(* PLC project PLC_DEV.project, CODESYS CODESYS V3.5 SP21 Patch 4 *)
(* stored: creationDateTime 1970-01-01T00:00:00, modificationDateTime 1970-01-01T00:00:00 *)

TYPE ST_IO_IN : STRUCT
  StartPB : BOOL;
  StopPB : BOOL;
  EStop : BOOL;
  LS_Extended : BOOL;
  LS_Retracted : BOOL;
  MotorFB : BOOL;
  TankLevel : REAL;  (* 0..100 % *)
  Pressure : REAL;
  ValvePosFB : REAL;  (* 0..100 % *)
END_STRUCT;
END_TYPE

TYPE ST_IO_OUT : STRUCT
  MotorRun : BOOL;
  Pump : BOOL;
  CylExtend : BOOL;
  CylRetract : BOOL;
  ValveCmd : REAL;  (* 0..100 % *)
  VFD_SpeedCmd : REAL;  (* 0..100 % *)
END_STRUCT;
END_TYPE

TYPE ST_IO : STRUCT
  In : ST_IO_IN;
  Out : ST_IO_OUT;
END_STRUCT;
END_TYPE

(* values of E_SIM_BOOL_MODE: FIXED: always FixedValue (or OverrideValue); TOGGLE: flips true/false every ChangeEvery; PULSE: true for PulseWidth every ChangeEvery *)

TYPE E_SIM_BOOL_MODE : (FIXED, TOGGLE, PULSE);
END_TYPE

(* values of E_SIM_INT_MODE: FIXED: fixed value; RAMP: add Increment every ChangeEvery; RANDOM: pseudo-random in range every ChangeEvery *)

TYPE E_SIM_INT_MODE : (FIXED, RAMP, RANDOM);
END_TYPE

TYPE E_RunMode : (DEV, STG, PROD);
END_TYPE

PROGRAM PLC_PRG
  VAR
    Boot : FB_ModeBoot;
    IOMan : FB_IO_Manager;
  END_VAR

                  // 1) Read ENV ONCE
Boot();

// 2) Route IO
IOMan(Mode := gMode, IO := gIO);

// 3) Control logic


// ---------------- Control Logic ----------------
IF gIO.In.EStop THEN
    gIO.Out.MotorRun := FALSE;
    gIO.Out.Pump := FALSE;
    gIO.Out.CylExtend := FALSE;
	gIO.Out.VFD_SpeedCmd := 0.0; // going back to 0
    gIO.Out.ValveCmd := 0.0;  // same here
ELSE
    IF gIO.In.StartPB THEN
        gIO.Out.MotorRun := TRUE;
        gIO.Out.Pump := TRUE;
        gIO.Out.VFD_SpeedCmd := 75.0; // Increase the speed 
        gIO.Out.ValveCmd := 15.0; // Valve command should be 15
    END_IF

    IF gIO.In.StopPB THEN
        gIO.Out.MotorRun := FALSE;
        gIO.Out.Pump := FALSE;
        gIO.Out.VFD_SpeedCmd := 0.0;
        gIO.Out.ValveCmd := 0.0;
    END_IF

    gIO.Out.CylExtend := gIO.Out.MotorRun;
    gIO.Out.CylRetract := NOT gIO.Out.MotorRun;
END_IF
                
END_PROGRAM

FUNCTION_BLOCK FB_IO_Prod
  VAR_IN_OUT
    IO : ST_IO;
  END_VAR

                  // ================= READ PROD INPUTS =================
// Map your physical / fieldbus / Modbus / MQTT inputs here
// Example:
// IO.In.StartPB      := TRUE;
// IO.In.StopPB       := DI_StopPB;
// IO.In.EStop        := DI_EStop;
// IO.In.LS_Extended  := DI_LS_Extended;
// IO.In.LS_Retracted := DI_LS_Retracted;
// IO.In.MotorFB      := DI_MotorFB;
//
// IO.In.TankLevel    := AI_TankLevel;
// IO.In.Pressure     := AI_Pressure;
// IO.In.ValvePosFB   := AI_ValvePosFB;

// ================= WRITE PROD OUTPUTS =================
// Example:
// DO_MotorRun     := IO.Out.MotorRun;
// DO_Pump         := IO.Out.Pump;
// DO_CylExtend    := IO.Out.CylExtend;
// DO_CylRetract   := IO.Out.CylRetract;
//
// AO_ValveCmd     := IO.Out.ValveCmd;
// AO_VFD_SpeedCmd := IO.Out.VFD_SpeedCmd;
                
END_FUNCTION_BLOCK

FUNCTION_BLOCK FB_IO_Manager
  VAR_INPUT
    Mode : E_RunMode;
  END_VAR
  VAR_IN_OUT
    IO : ST_IO;
  END_VAR
  VAR
    Sim : FB_IO_SIM;
    Prod : FB_IO_PROD;
  END_VAR

                  // DEV + STG = simulated IO
IF (Mode = E_RunMode.DEV) OR (Mode = E_RunMode.STG) THEN
    Sim(IO := IO);
ELSE
    Prod(IO := IO);
END_IF

                
END_FUNCTION_BLOCK

FUNCTION_BLOCK FB_ModeBoot
  VAR_OUTPUT
    Done : BOOL;
  END_VAR
  VAR
    init : BOOL;
    outBuf : STRING(64);
    res : DINT;
    n : DINT;
  END_VAR

                  IF Done THEN RETURN; END_IF
IF NOT init THEN
    init := TRUE;

    gMode := E_RunMode.PROD;   // safe default
    outBuf := '';

    n := SysProcessExecuteCommand2(
        pszCommand := '/usr/bin/head -c 4 /conf/codesyscontrol/env.txt',
        pszStdOut := outBuf,
        udiStdOutLen := SIZEOF(outBuf),
        pResult := ADR(res)
    );

    IF n >= 3 THEN
        IF (LEFT(outBuf, 3) = 'dev') OR (LEFT(outBuf, 3) = 'DEV') THEN
            gMode := E_RunMode.DEV;

        ELSIF (LEFT(outBuf, 3) = 'stg') OR (LEFT(outBuf, 3) = 'STG') THEN
            gMode := E_RunMode.STG;

        ELSIF (LEFT(outBuf, 4) = 'prod') OR (LEFT(outBuf, 4) = 'PROD') THEN
            gMode := E_RunMode.PROD;
        END_IF
    END_IF

    Done := TRUE;
END_IF


                
END_FUNCTION_BLOCK

FUNCTION_BLOCK FB_SimInt_Gen
  VAR_INPUT
    Enable : BOOL := TRUE;
    Mode : E_SIM_INT_MODE := E_SIM_INT_MODE.RAMP;
    MinValue : INT := 0;
    MaxValue : INT := 100;
    Increment : INT := 1;  (* used by RAMP *)
    ChangeEvery : TIME := TIME#200ms;
    Wrap : BOOL := TRUE;  (* RAMP behavior: wrap or clamp *)
    FixedValue : INT := 0;
    OverrideEn : BOOL := FALSE;
    OverrideValue : INT := 0;
  END_VAR
  VAR_OUTPUT
    Value : INT;
  END_VAR
  VAR
    tPeriod : TON;
    seedInt : INT := 12345;  (* random seed kept as INT only *)
    span : INT;
    nextVal : INT;
    tmp : INT;
  END_VAR

                  // ---------- guards ----------
IF NOT Enable THEN
    Value := MinValue;
    RETURN;
END_IF

IF OverrideEn THEN
    Value := OverrideValue;
    RETURN;
END_IF

IF MaxValue < MinValue THEN
    Value := MinValue;
    RETURN;
END_IF

// ---------- timing ----------
tPeriod(IN := TRUE, PT := ChangeEvery);
IF NOT tPeriod.Q THEN
    RETURN;
END_IF
tPeriod(IN := FALSE); // restart timer

// ---------- mode ----------
CASE Mode OF

E_SIM_INT_MODE.FIXED:
    Value := FixedValue;

E_SIM_INT_MODE.RAMP:
    nextVal := Value + Increment;

    IF Wrap THEN
        span := MaxValue - MinValue + 1;
        IF span <= 0 THEN span := 1; END_IF
        WHILE nextVal > MaxValue DO
            nextVal := nextVal - span;
        END_WHILE
        WHILE nextVal < MinValue DO
            nextVal := nextVal + span;
        END_WHILE
    ELSE
        IF nextVal > MaxValue THEN nextVal := MaxValue; END_IF
        IF nextVal < MinValue THEN nextVal := MinValue; END_IF
    END_IF

    Value := nextVal;

E_SIM_INT_MODE.RANDOM:
    // simple INT LCG (stays in INT domain)
    seedInt := seedInt * 109 + 89;

    // make it non-negative
    IF seedInt < 0 THEN
        seedInt := -seedInt;
    END_IF

    span := MaxValue - MinValue + 1;
    IF span <= 0 THEN span := 1; END_IF

    // reduce into 0..span-1 using subtraction (no MOD needed)
    tmp := seedInt;
    WHILE tmp >= span DO
        tmp := tmp - span;
    END_WHILE

    Value := MinValue + tmp;

END_CASE
                
END_FUNCTION_BLOCK

FUNCTION_BLOCK FB_SimBool_Gen
  VAR_INPUT
    Enable : BOOL := TRUE;
    Mode : E_SIM_BOOL_MODE := E_SIM_BOOL_MODE.TOGGLE;
    ChangeEvery : TIME := TIME#2s0ms;
    PulseWidth : TIME := TIME#150ms;
    FixedValue : BOOL := FALSE;
    OverrideEn : BOOL := FALSE;
    OverrideValue : BOOL := FALSE;
  END_VAR
  VAR_OUTPUT
    Value : BOOL;
  END_VAR
  VAR
    tPeriod : TON;
    tPulse : TON;
    state : BOOL := FALSE;
  END_VAR

                  IF NOT Enable THEN
    Value := FALSE;
    RETURN;
END_IF

IF OverrideEn THEN
    Value := OverrideValue;
    RETURN;
END_IF

CASE Mode OF

E_SIM_BOOL_MODE.FIXED:
    Value := FixedValue;

E_SIM_BOOL_MODE.TOGGLE:
    tPeriod(IN := TRUE, PT := ChangeEvery);
    IF tPeriod.Q THEN
        state := NOT state;
        tPeriod(IN := FALSE);
    END_IF
    Value := state;

E_SIM_BOOL_MODE.PULSE:
    tPeriod(IN := TRUE, PT := ChangeEvery);
    IF tPeriod.Q THEN
        tPulse(IN := TRUE, PT := PulseWidth);
        tPeriod(IN := FALSE);
    END_IF
    tPulse(IN := tPulse.IN, PT := PulseWidth);
    Value := tPulse.Q;

END_CASE

                
END_FUNCTION_BLOCK

FUNCTION_BLOCK FB_IO_Sim
  VAR_IN_OUT
    IO : ST_IO;
  END_VAR
  VAR
    StartPB_Sim : FB_SimBool_Gen;
    StartPB_Value : BOOL;
    TankLevel_Sim : FB_SimInt_Gen;
  END_VAR

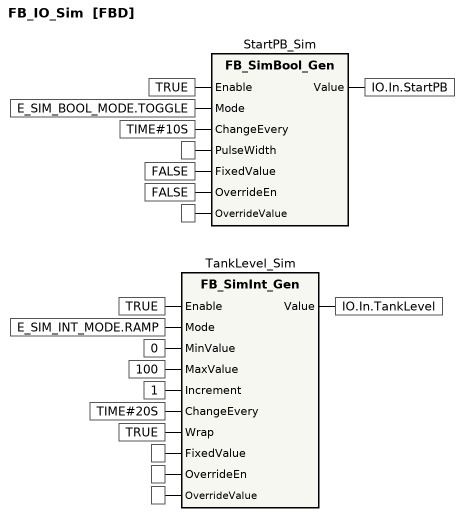
(* FBD diagram, written out as Structured Text *)
StartPB_Sim(Enable := TRUE, Mode := E_SIM_BOOL_MODE.TOGGLE, ChangeEvery := TIME#10S, PulseWidth := , FixedValue := FALSE, OverrideEn := FALSE, OverrideValue := );
IO.In.StartPB := StartPB_Sim.Value;
TankLevel_Sim(Enable := TRUE, Mode := E_SIM_INT_MODE.RAMP, MinValue := 0, MaxValue := 100, Increment := 1, ChangeEvery := TIME#20S, Wrap := TRUE, FixedValue := , OverrideEn := , OverrideValue := );
IO.In.TankLevel := TankLevel_Sim.Value;
END_FUNCTION_BLOCK

CONFIGURATION Application
  RESOURCE Application ON PLC
    VAR_GLOBAL  (* GVL_IO *)
      gIO : ST_IO;
      gIsDev : BOOL := FALSE;
      gMode : E_RunMode := E_RunMode.PROD;
    END_VAR
    TASK MainTask(INTERVAL := T#20ms, PRIORITY := 1);
    PROGRAM PLC_PRG WITH MainTask : PLC_PRG;
  END_RESOURCE
END_CONFIGURATION
